SUBAPPLICATION Uebung_012f_sub (* Numeric Value Input PHYS und Speichern NVS mit Subapp *)
  (* Standard: 61499-2; Description: Copyright (c) 2023 Meisterschulen am Ostbahnhof This program and the accompanying materials are made available under the terms of the Eclipse Public License 2.0 which is available at https://www.eclipse.org/legal/epl-2.0/ SPDX-License-Identifier: EPL-2.0 *)
  (* Version 1.0, 2023-10-31, Franz Höpfinger, Meisterschulen am Ostbahnhof, initial API and implementation and/or initial documentation *)
  PACKAGE Uebungen;
  IMPORT isobus::UT::Q::const::IDs::ID_NULL;
  IMPORT logiBUS::utils::conversion::phys::NumericObjectPool_S;
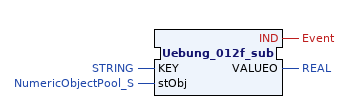
  EVENT_OUTPUT
    IND;
  END_EVENT
  VAR_INPUT
    KEY : STRING; (* Key name. *)
    stObj : logiBUS::utils::conversion::phys::NumericObjectPool_S := (u16ObjId := ID_NULL, r32Scale := 1.0, i32Offset := 0, u8Decimals := 0);
  END_VAR
  VAR_OUTPUT
    VALUEO : REAL;
  END_VAR
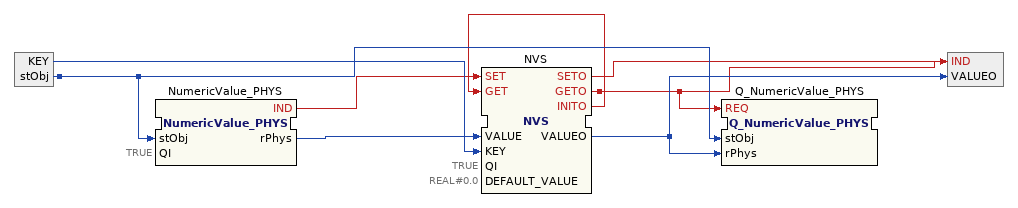
  FBS
    NumericValue_PHYS : isobus::UT::io::NumericValue::NumericValue_PHYS(QI := TRUE);
    NVS : logiBUS::storage::esp32_nvs::NVS(QI := TRUE, DEFAULT_VALUE := REAL#0.0);
    Q_NumericValue_PHYS : isobus::UT::Q::Q_NumericValue_PHYS;
  END_FBS
  EVENT_CONNECTIONS
    NumericValue_PHYS.IND TO NVS.SET;
    NVS.SETO TO IND;
    NVS.GETO TO Q_NumericValue_PHYS.REQ;
    NVS.GETO TO IND;
    NVS.INITO TO NVS.GET;
  END_CONNECTIONS
  DATA_CONNECTIONS
    NumericValue_PHYS.rPhys TO NVS.VALUE;
    stObj TO Q_NumericValue_PHYS.stObj;
    KEY TO NVS.KEY;
    NVS.VALUEO TO Q_NumericValue_PHYS.rPhys;
    NVS.VALUEO TO VALUEO;
    stObj TO NumericValue_PHYS.stObj;
  END_CONNECTIONS
END_SUBAPPLICATION
